FUNCTION_BLOCK MaintenanceCounter
VAR_INPUT
	 CU      : BOOL; (* Count Up *)
     RESET   : BOOL; (* Reset Counter to 0 *)
     PV      : DWORD; (* Counter Limit *)
END_VAR
VAR_OUTPUT
	Q       : BOOL; (* Counter reached the Limit *)
    CV      : DWORD; (* Current Counter Value *)
END_VAR
VAR PERSISTENT
	RisingEdge : R_TRIG;
	CurrentValue : DWORD;
END_VAR

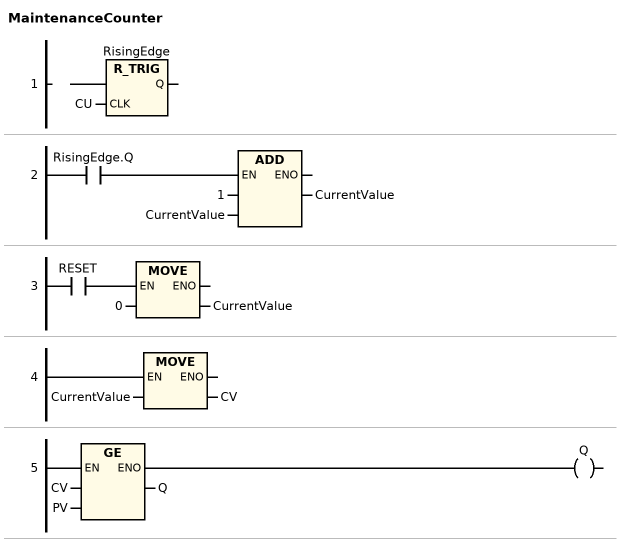
// NETWORK 1
RisingEdge(CLK := CU); // R_TRIG

// NETWORK 2
IF RisingEdge.Q THEN CurrentValue := 1 + CurrentValue; END_IF

// NETWORK 3
IF RESET THEN CurrentValue := 0; END_IF

// NETWORK 4
CV := CurrentValue;

// NETWORK 5
Q := CV >= PV;
Q := TRUE;

END_FUNCTION_BLOCK

(* stored: Version 1.1.0.1, ProductVersion 3.1.4020.12
   POU MaintenanceCounter: Id {9ba54e98-d73e-475d-a5ad-d03f6c4a8825}, SpecialFunc None *)
